# EPICS StreamDevice protocol: tti355Sup/tti355.proto
OutTerminator = "\n";
InTerminator = "\r\n";

# Set the output voltage
setVoltage {
    out "V %f";
    @init{ out "V?"; in "V%f"; }
}

# Get the output voltage
getSetpointVoltage{
    out "V?";
    in "V%f";
}

# Get the output voltage
getActualVoltage {
    out "VO?";
    in "V%f";
}

getIDN {
    out "*IDN?";
    in "%#s";
    ExtraInput = Ignore;
}

# Set the output current
setCurrent {
    out "I %f";
    @init{ out "I?"; in "I%f"; }
}

# Get the output current
getSetpointCurrent {
    out "I?";
    in "I%f";
}

# Get the actual output current
getActualCurrent {
    out "IO?";
    in "I%f";
}

# Set the output state
setOutput
    {
    out "%{OFF|ON}";
    }

# Get the output state
getOutput
    {
    out "OUT?";
    in "OUT %{OFF|ON}";
    }

# Get the error register
getError
    {
    out "ERR?";
    in "ERR %d";
    }

reset
    {
    out "*RST";
    }

# Get the output mode status
# this reflects whether the supply is voltage or current limiting (automatically switched)
getMode
    {
    out "M?";
    in "M C%{V|I}";
    }

cmd {
    out "\$1";
}

setD {
    out "\$1 %d";
}
getD {
    out "\$1?";
    in "%d";
    ExtraInput = Ignore;
}
